FUNCTION_BLOCK USINT2USINT (* Basic Function Block Type *)
  (* Standard: 61499-2; Description: Copyright (c) 2006 Profactor GmbH This program and the accompanying materials are made available under the terms of the Eclipse Public License 2.0 which is available at https://www.eclipse.org/legal/epl-2.0/ SPDX-License-Identifier: EPL-2.0 *)
  (* Version 1.0, 2006-11-14, Thomas Strasser, PROFACTOR GmbH, initial API and implementation and/or initial documentation *)
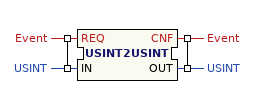
  EVENT_INPUT
    REQ WITH IN; (* Normal Execution Request *)
  END_EVENT
  EVENT_OUTPUT
    CNF WITH OUT; (* Execution Confirmation *)
  END_EVENT
  VAR_INPUT
    IN : USINT; (* Input event qualifier *)
  END_VAR
  VAR_OUTPUT
    OUT : USINT; (* Output event qualifier *)
  END_VAR
END_FUNCTION_BLOCK
